# EPICS autosave request: bpmApp/Db/SIS8300bpmN_settings.req
$(P)$(R)ThrXPosLow
$(P)$(R)ThrXPosHigh
$(P)$(R)ThrYPosLow
$(P)$(R)ThrYPosHigh
$(P)$(R)ThrMagnitude
$(P)$(R)ThrSelect
$(P)$(R)IlkControl
